FUNCTION_BLOCK FB_PWM_1
VAR_INPUT
	pwmCycleTime 		: TIME := T#10S;
	pwmDutyCycle		: REAL := 0.5;
	reset				: BOOL := FALSE;
END_VAR
VAR_OUTPUT
	Q					: BOOL := FALSE;
END_VAR
VAR
	pwmTimeInMs			: REAL	:= 0;
	pwmTimer			: FB_TON;
	dutyCycleInMs		: TIME;
	test				: INT;
	internalReset 		: BOOL := FALSE;
	goHigh				: BOOL := FALSE;
	
	temp1				: REAL;
	temp2				: DINT;
	temp3				: REAL;
	temp4				: REAL;
	
END_VAR

IF pwmDutyCycle < 0 THEN
	pwmDutyCycle := 0.0;
END_IF

IF reset OR internalReset THEN
	pwmTimer(IN:= FALSE);
	reset := FALSE;
	internalReset := FALSE;
	IF goHigh THEN
		temp1 := (1.0-pwmDutyCycle);
		temp2 := REAL_TO_DINT(pwmTimeInMs*(1.0-pwmDutyCycle));
		dutyCycleInMs := DINT_TO_TIME(REAL_TO_DINT(pwmTimeInMs*(1.0-pwmDutyCycle)));
		goHigh := FALSE;
	ELSE
		temp1 := (1.0-pwmDutyCycle);
		temp2 := REAL_TO_DINT(pwmTimeInMs*(1.0-pwmDutyCycle));
		dutyCycleInMs := DINT_TO_TIME(REAL_TO_DINT(pwmTimeInMs*pwmDutyCycle));
	END_IF
ELSE
	pwmTimeInMs := DINT_TO_REAL(TIME_TO_DINT(pwmCycleTime));
	IF Q THEN
		(* high  --> running falling timer *)
		(*dutyCycleInMs := DINT_TO_TIME(REAL_TO_DINT(pwmTimeInMs*pwmDutyCycle));*)
		pwmTimer(IN:=TRUE, PT:=dutyCycleInMs);
		IF pwmTimer.Q THEN
			internalReset := TRUE;
			Q := FALSE;
			goHigh := TRUE;
			pwmTimer(IN:=FALSE);
		END_IF		
	ELSE
		(* low --> running rising timer *)
		pwmTimer(IN:=TRUE, PT:=dutyCycleInMs);
		IF pwmTimer.Q THEN
			internalReset := TRUE;
			Q := TRUE;
			pwmTimer(IN:=FALSE);
		END_IF		
	END_IF
END_IF

END_FUNCTION_BLOCK

(* stored: Version 1.1.0.1, ProductVersion 3.1.4022.12
   POU FB_PWM_1: Id {b4123095-a844-4446-8e1e-c07c87a44182}, SpecialFunc None *)
